Staubli VAL3: cvIn.pjx

--- cvIn.pjx ---
Parameters version=s7.6.2 stackSize=5000 millimeterUnit=true
Program file=checkTrackArea.pgx
Program file=conveyor.pgx
Program file=create.pgx
Program file=disableQueue.pgx
Program file=enableQueue.pgx
Program file=fillQueue.pgx
Program file=flushQueue.pgx
Program file=getConvFrame.pgx
Program file=getDetectDist.pgx
Program file=getDetectFrame.pgx
Program file=getDistance.pgx
Program file=getErrorMessage.pgx
Program file=getNextID.pgx
Program file=getObjectData.pgx
Program file=getObjectLatch.pgx
Program file=getObjectOffset.pgx
Program file=getObjectPos.pgx
Program file=getStatus.pgx
Program file=getTravelDist.pgx
Program file=init.pgx
Program file=kill.pgx
Program file=releaseObject.pgx
Program file=removePart.pgx
Program file=reset.pgx
Program file=setCalibrating.pgx
Program file=setConveyor.pgx
Program file=setObjectInUse.pgx
Program file=start.pgx
Program file=stop.pgx
Program file=teach.pgx
Program file=whichObjectUsed.pgx
Data file=cvIn.dtx
Library alias=cfg path=Disk://Tracking/config/config.pjx autoload=true password=
Library alias=det path=Disk://Tracking/Templates/GenericDetect/GenericDetect.pjx autoload=false password=
Library alias=enc path=Disk://Tracking/Templates/GenericEnc/GenericEnc.pjx autoload=false password=
Library alias=geometry path=Disk://Tracking/Templates/Geometry/Geometry.pjx autoload=false password=
Library alias=swap path=Disk://Tracking/Swap/Swap.pjx autoload=true password=
Library alias=ut path=Disk://Tracking/Tools/util/util.pjx autoload=true password=
Library alias=lang path=Disk://Tracking/language/english/english.pjx autoload=true password=
Library alias=out path=Disk://Tracking/io/outputs/outputs.pjx autoload=true password=

--- cvIn.dtx ---
bool bClockEnabled = true
bool bEnableQueuing = true
bool bInit = true
public bool bLOG = true
public bool bLinear = true
bool bLockQueueAcces
bool bResetConv
public bool bUseUserCenter
public bool bUseUserLimit
dio doClock = {link=BasicIO-1\%Q0}
public frame fConveyor = {x=365.904087, y=326.91934, z=-82.602337, rx=-0.010861, ry=-0.059106, rz=0.004608, fatherId=world[0]}
public frame fDetection = {x=392.598601, y=461.346273, z=-82.976862, rx=0.205045, ry=0.617271, rz=0.011036, fatherId=world[0]}
num nA1 = -1.427414
num nA2 = -1.428787
num nAddedToQueue
num nB1
num nB2 = 436.58822
num nBoundaryDwn
num nBoundaryUp
public num nBufferSize = 100
public num nCalibratedDist
num nCalibratedID = -99
public num nClockPeriod = 210
public num nConveyorSpeed = 495.277368
num nDEFAULTID = -99
num nDETECT_OVR = 11
public num nDetection2Rob = 945.961992
public num nENCRESOLUTION = 2000
public num nENCSCALEFACTOR = 0.7207
num nEncLatchedVal[100]
num nErrVal[4]
public num nFirDelay = 0.004
public num nFirOrdre = 20
num nFirTime = 0.04
num nIdxCalib
num nIdxPull
num nIdxPush
public num nLatchLockDist
num nNumbOfUser[100]
num nPUSH_NEGATIVE = 10
public num nPosMatchTol = 50
num nQueueID[100]
  [0] = -99
  [1] = -99
  [2] = -99
  [3] = -99
  [4] = -99
  [5] = -99
  [6] = -99
  [7] = -99
  [8] = -99
  [9] = -99
  [10] = -99
  [11] = -99
  [12] = -99
  [13] = -99
  [14] = -99
  [15] = -99
  [16] = -99
  [17] = -99
  [18] = -99
  [19] = -99
  [20] = -99
  [21] = -99
  [22] = -99
  [23] = -99
  [24] = -99
  [25] = -99
  [26] = -99
  [27] = -99
  [28] = -99
  [29] = -99
  [30] = -99
  [31] = -99
  [32] = -99
  [33] = -99
  [34] = -99
  [35] = -99
  [36] = -99
  [37] = -99
  [38] = -99
  [39] = -99
  [40] = -99
  [41] = -99
  [42] = -99
  [43] = -99
  [44] = -99
  [45] = -99
  [46] = -99
  [47] = -99
  [48] = -99
  [49] = -99
  [50] = -99
  [51] = -99
  [52] = -99
  [53] = -99
  [54] = -99
  [55] = -99
  [56] = -99
  [57] = -99
  [58] = -99
  [59] = -99
  [60] = -99
  [61] = -99
  [62] = -99
  [63] = -99
  [64] = -99
  [65] = -99
  [66] = -99
  [67] = -99
  [68] = -99
  [69] = -99
  [70] = -99
  [71] = -99
  [72] = -99
  [73] = -99
  [74] = -99
  [75] = -99
  [76] = -99
  [77] = -99
  [78] = -99
  [79] = -99
  [80] = -99
  [81] = -99
  [82] = -99
  [83] = -99
  [84] = -99
  [85] = -99
  [86] = -99
  [87] = -99
  [88] = -99
  [89] = -99
  [90] = -99
  [91] = -99
  [92] = -99
  [93] = -99
  [94] = -99
  [95] = -99
  [96] = -99
  [97] = -99
  [98] = -99
  [99] = -99
num nStatus
num nSysCycleTime = 0.002
num nTmpEncLatched[10]
  [0] = 4878005.31
  [1] = 4869824.31
  [2] = 4741503.57
num nTmpID[10]
  [0] = 1
  [1] = 1
  [2] = 1
public num nTrackWinHeight = 500
num nWinDownStream
num nWinUpStream
pointRs pObjectRS = {fatherId=world[0]}
pointRx pObject = {fatherId=world[0]}
public string sClockSigName = "bOut0"
string sConvNum = "CNV0"
public string sConveyorName = "cvIn"
public string sDetectionLib = "PointGrey"
public string sDwnLimSigName = "none"
public string sEncoderLib = "D_ABZ_00"
string sErrMsgList[12]
  [0] = "Success"
  [1] = "No object available (ID=*)"
  [3] = "The encoder library is not started yet."
  [4] = "The detection library is not started yet."
  [6] = "Run-time error from Conveyor library in task called *\../*. Error code is *"
  [7] = "Run-time error from Encoder library. Error code is *"
  [8] = "Run-time error from Detection library. Error code is *"
  [10] = "Warning, object with negative ID cannot be pushed into conveyor's queue"
  [11] = "Warning, detection overrun."
string sErrorMessage = "No message pending"
public string sGeometryLib = "GeometryRS"
string sMsg
string sTASK[3]
  [0] = "conveyor"
  [1] = "encoder"
  [2] = "detect"
public string sUpLimSigName = "none"
trsf trBoundaryDwn[2]
  [0] = {x=305.565702, rx=-179.989134, ry=-0.059105, rz=88.399965}
  [1] = {x=118.089887, y=267.862957, z=0.515773, rx=-179.989134, ry=-0.059105, rz=65.426002}
trsf trBoundaryUp[2]
  [0] = {rx=-179.989134, ry=-0.059105, rz=58.053225}
  [1] = {x=-187.656083, y=267.862957, rx=-179.989134, ry=-0.059105, rz=32.698528}
trsf trDEFAULT = {x=5, y=4, z=3, rx=2, ry=1}
trsf trDetectedCoord[100]
  [0] = {x=5, y=4, z=3, rx=2, ry=1}
  [1] = {x=5, y=4, z=3, rx=2, ry=1}
  [2] = {x=5, y=4, z=3, rx=2, ry=1}
  [3] = {x=5, y=4, z=3, rx=2, ry=1}
  [4] = {x=5, y=4, z=3, rx=2, ry=1}
  [5] = {x=5, y=4, z=3, rx=2, ry=1}
  [6] = {x=5, y=4, z=3, rx=2, ry=1}
  [7] = {x=5, y=4, z=3, rx=2, ry=1}
  [8] = {x=5, y=4, z=3, rx=2, ry=1}
  [9] = {x=5, y=4, z=3, rx=2, ry=1}
  [10] = {x=5, y=4, z=3, rx=2, ry=1}
  [11] = {x=5, y=4, z=3, rx=2, ry=1}
  [12] = {x=5, y=4, z=3, rx=2, ry=1}
  [13] = {x=5, y=4, z=3, rx=2, ry=1}
  [14] = {x=5, y=4, z=3, rx=2, ry=1}
  [15] = {x=5, y=4, z=3, rx=2, ry=1}
  [16] = {x=5, y=4, z=3, rx=2, ry=1}
  [17] = {x=5, y=4, z=3, rx=2, ry=1}
  [18] = {x=5, y=4, z=3, rx=2, ry=1}
  [19] = {x=5, y=4, z=3, rx=2, ry=1}
  [20] = {x=5, y=4, z=3, rx=2, ry=1}
  [21] = {x=5, y=4, z=3, rx=2, ry=1}
  [22] = {x=5, y=4, z=3, rx=2, ry=1}
  [23] = {x=5, y=4, z=3, rx=2, ry=1}
  [24] = {x=5, y=4, z=3, rx=2, ry=1}
  [25] = {x=5, y=4, z=3, rx=2, ry=1}
  [26] = {x=5, y=4, z=3, rx=2, ry=1}
  [27] = {x=5, y=4, z=3, rx=2, ry=1}
  [28] = {x=5, y=4, z=3, rx=2, ry=1}
  [29] = {x=5, y=4, z=3, rx=2, ry=1}
  [30] = {x=5, y=4, z=3, rx=2, ry=1}
  [31] = {x=5, y=4, z=3, rx=2, ry=1}
  [32] = {x=5, y=4, z=3, rx=2, ry=1}
  [33] = {x=5, y=4, z=3, rx=2, ry=1}
  [34] = {x=5, y=4, z=3, rx=2, ry=1}
  [35] = {x=5, y=4, z=3, rx=2, ry=1}
  [36] = {x=5, y=4, z=3, rx=2, ry=1}
  [37] = {x=5, y=4, z=3, rx=2, ry=1}
  [38] = {x=5, y=4, z=3, rx=2, ry=1}
  [39] = {x=5, y=4, z=3, rx=2, ry=1}
  [40] = {x=5, y=4, z=3, rx=2, ry=1}
  [41] = {x=5, y=4, z=3, rx=2, ry=1}
  [42] = {x=5, y=4, z=3, rx=2, ry=1}
  [43] = {x=5, y=4, z=3, rx=2, ry=1}
  [44] = {x=5, y=4, z=3, rx=2, ry=1}
  [45] = {x=5, y=4, z=3, rx=2, ry=1}
  [46] = {x=5, y=4, z=3, rx=2, ry=1}
  [47] = {x=5, y=4, z=3, rx=2, ry=1}
  [48] = {x=5, y=4, z=3, rx=2, ry=1}
  [49] = {x=5, y=4, z=3, rx=2, ry=1}
  [50] = {x=5, y=4, z=3, rx=2, ry=1}
  [51] = {x=5, y=4, z=3, rx=2, ry=1}
  [52] = {x=5, y=4, z=3, rx=2, ry=1}
  [53] = {x=5, y=4, z=3, rx=2, ry=1}
  [54] = {x=5, y=4, z=3, rx=2, ry=1}
  [55] = {x=5, y=4, z=3, rx=2, ry=1}
  [56] = {x=5, y=4, z=3, rx=2, ry=1}
  [57] = {x=5, y=4, z=3, rx=2, ry=1}
  [58] = {x=5, y=4, z=3, rx=2, ry=1}
  [59] = {x=5, y=4, z=3, rx=2, ry=1}
  [60] = {x=5, y=4, z=3, rx=2, ry=1}
  [61] = {x=5, y=4, z=3, rx=2, ry=1}
  [62] = {x=5, y=4, z=3, rx=2, ry=1}
  [63] = {x=5, y=4, z=3, rx=2, ry=1}
  [64] = {x=5, y=4, z=3, rx=2, ry=1}
  [65] = {x=5, y=4, z=3, rx=2, ry=1}
  [66] = {x=5, y=4, z=3, rx=2, ry=1}
  [67] = {x=5, y=4, z=3, rx=2, ry=1}
  [68] = {x=5, y=4, z=3, rx=2, ry=1}
  [69] = {x=5, y=4, z=3, rx=2, ry=1}
  [70] = {x=5, y=4, z=3, rx=2, ry=1}
  [71] = {x=5, y=4, z=3, rx=2, ry=1}
  [72] = {x=5, y=4, z=3, rx=2, ry=1}
  [73] = {x=5, y=4, z=3, rx=2, ry=1}
  [74] = {x=5, y=4, z=3, rx=2, ry=1}
  [75] = {x=5, y=4, z=3, rx=2, ry=1}
  [76] = {x=5, y=4, z=3, rx=2, ry=1}
  [77] = {x=5, y=4, z=3, rx=2, ry=1}
  [78] = {x=5, y=4, z=3, rx=2, ry=1}
  [79] = {x=5, y=4, z=3, rx=2, ry=1}
  [80] = {x=5, y=4, z=3, rx=2, ry=1}
  [81] = {x=5, y=4, z=3, rx=2, ry=1}
  [82] = {x=5, y=4, z=3, rx=2, ry=1}
  [83] = {x=5, y=4, z=3, rx=2, ry=1}
  [84] = {x=5, y=4, z=3, rx=2, ry=1}
  [85] = {x=5, y=4, z=3, rx=2, ry=1}
  [86] = {x=5, y=4, z=3, rx=2, ry=1}
  [87] = {x=5, y=4, z=3, rx=2, ry=1}
  [88] = {x=5, y=4, z=3, rx=2, ry=1}
  [89] = {x=5, y=4, z=3, rx=2, ry=1}
  [90] = {x=5, y=4, z=3, rx=2, ry=1}
  [91] = {x=5, y=4, z=3, rx=2, ry=1}
  [92] = {x=5, y=4, z=3, rx=2, ry=1}
  [93] = {x=5, y=4, z=3, rx=2, ry=1}
  [94] = {x=5, y=4, z=3, rx=2, ry=1}
  [95] = {x=5, y=4, z=3, rx=2, ry=1}
  [96] = {x=5, y=4, z=3, rx=2, ry=1}
  [97] = {x=5, y=4, z=3, rx=2, ry=1}
  [98] = {x=5, y=4, z=3, rx=2, ry=1}
  [99] = {x=5, y=4, z=3, rx=2, ry=1}
trsf trTmp[10]
  [0] = {x=-13.6, y=13.6, rz=90}
  [1] = {x=-105.5, y=-8.6, rz=91}
  [2] = {x=-185.6, y=-3.4, rz=87.4}

--- conveyor.pgx ---
program conveyor()
  local bool l_bLatched
  local bool l_bLock
  local bool l_bMemoCalib
  local num l_nDelayEnLatch
  local num l_nEncEnaLatVal
  local num l_nEncLatchVal
  local num l_nEncValue
  local num l_nLatchLocked
  local num l_nNumOfObject
  local num l_nStepFill
  local num l_nTimeLatched
  local num l_nTrigger
begin
  //
  //----------------------------------------------------------------
  l_nEncEnaLatVal=l_nEncLatchVal=l_nEncValue
  l_bMemoCalib=det:bCalibrating
  //
  //--- Enable latch feature of the encoder library
  enc:bLatchEnabled=true
  if bClockEnabled
    l_nStepFill=-1
  else
    l_nStepFill=0
  endIf
  l_nTimeLatched=clock()
  //*****
  //
  // Initializing the output to start if it's used
  if bClockEnabled
    // If position capture OUTPUT occurs on falling edge
    // CHANGE the logic of the output doClock at all lines of this program.
    // false-->true / true-->false
    doClock=false
  endIf
  // waiting the task's detection is running
  wait(det:bTaskDetOK)
  //****   MAIN LOOP
  while true
    //--- Read instantaneous encoder value
    l_nEncValue=aioGet(enc:aiEncCurrentPos)
    //
    //*****  CLOCK SECTION
    l_nLatchLocked=sel(bClockEnabled,max(2*nClockPeriod/3,nLatchLockDist),nLatchLockDist)
    // Check if feature is enabled
    if bClockEnabled
      // If trigger OFF, and If the conveyor has moved more than the trigger perriod
      if (doClock==false) and abs((l_nEncValue-l_nEncEnaLatVal)*nENCSCALEFACTOR)>nClockPeriod
        // If system ready, set trigger
        // Else, set Status in overrun
        if l_nStepFill==-1
          l_nStepFill=0
          doClock=true
          l_nTrigger=l_nTrigger+1
          logMsg("trigger num: "+toString("",l_nTrigger)+" :"+toString("0.2",clock())+" s")
          logMsg("trigger: "+toString(".2",(l_nEncValue-l_nEncEnaLatVal)*nENCSCALEFACTOR)+" mm")
          l_nEncEnaLatVal=l_nEncValue
          if bAnd(cfg:nLog,cfg:nLOGDETECT)==cfg:nLOGDETECT and bLOG
            ? sConvNum+"(conveyor)>>Set trigger. Clock :"+toString(".2",clock())
          endIf
        elseIf nStatus!=2
          // Warning, detection overrun. Object(s) wont been queued
          if bAnd(cfg:nLog,cfg:nLOGDETECT)==cfg:nLOGDETECT and bLOG
            ? sConvNum+"(conveyor)>>Detection Overrun : Cannot set trigger on time. Clock :"+toString(".2",clock())
          endIf
          nStatus=2
          sErrorMessage=sErrMsgList[nDETECT_OVR]
        endIf
      endIf
      // If trigger ON, and If the conveyor has move more than half of the trigger period
      // reset trigger
      if (doClock==true) and abs((l_nEncValue-l_nEncEnaLatVal)*nENCSCALEFACTOR)>nClockPeriod/2
        doClock=false
      endIf
    endIf
    //
    //*****  CONVEYOR SECTION
    if left(sDetectionLib,6)=="Socket" and !det:bCalibrating
      // When working with the detection library "Socket" and the conveyor
      //  isn't calibrating the distance from the sensor, the encoder
      //  latched value is given by the "Socket" and the encoder library is
      //  not used.
      l_bLatched=true
      l_nEncLatchVal=0
      if l_nStepFill==0
        l_nStepFill=1
      endIf
    else
      // Reinitialize conveyor sequence when detection library "Socket"
      //  goes into Calibration Mode.
      if left(sDetectionLib,6)=="Socket" and det:bCalibrating and !l_bMemoCalib
        l_nStepFill=0
        det:nNumOfPart=-1
      endIf
      // Use the encoder library to get the encoder latched value.
      // Check if latch occured
      call enc:isLatched(l_bLatched)
      // If part latched, get encoder latched value.
      // Else, re-enable latching at the encoder library
      if l_bLatched==true
        logMsg("getLatched: "+toString(".2",clock())+" s")
        det:nNumOfPart=-1
        delay(0)
        call enc:resetLatch()
        if bAnd(cfg:nLog,cfg:nLOGDETECT)==cfg:nLOGDETECT and bLOG
          ? sConvNum+"(conveyor)>>Object latched detected. Clock :"+toString(".2",clock())
        endIf
        //
        // Start timer for re-enabling latch feature
        l_nDelayEnLatch=clock()
        //
        // If system ready, get encoder latched value.
        // Else, overrun for external latch
        if l_nStepFill==0
          l_nStepFill=1
          l_bLock=false
          // Get encoder latched value
          call enc:getValue(true,l_nEncLatchVal)
          // Disable latch feature of the encoder library until conveyor has moved
          // the distance defined by the user (variable nLatchLockDist)
          enc:bLatchEnabled=false
          // Record clock of Latch
          l_nTimeLatched=clock()
          //
          //Overrun for external latch
        elseIf !bClockEnabled and nStatus!=2
          // Warning, detection overrun. Object(s) wont been queued
          if bAnd(cfg:nLog,cfg:nLOGDETECT)==cfg:nLOGDETECT and bLOG
            ? sConvNum+"(conveyor)>>Detection Overrun : System not ready to latch again."
          endIf
          nStatus=2
          sErrorMessage=sErrMsgList[nDETECT_OVR]
        endIf
      else
        // wait a while before re-enabling the latch feature
        if clock()-l_nDelayEnLatch>0.02
          // Latch feature not enabled
          if (enc:bLatchEnabled==false)
            // Check conveyor's advance
            if abs((l_nEncValue-l_nEncLatchVal)*nENCSCALEFACTOR)>=l_nLatchLocked
              enc:bLatchEnabled=true
            endIf
          endIf
        endIf
      endIf
    endIf
    l_bMemoCalib=det:bCalibrating
    //
    //--- Poll detection library
    if bEnableQueuing==true
      switch l_nStepFill
        // Poll detection lib for number of detected objects
        case 1
          if l_bLock==false
            if bAnd(cfg:nLog,cfg:nLOGDETECT)==cfg:nLOGDETECT and bLOG
              ? sConvNum+"(conveyor)>>Reading number of detected objects"
            endIf
            l_bLock=true
          endIf
          //
          if l_bLock==true
            call det:isDetected(l_nNumOfObject)
            if (l_nNumOfObject>=0)
              l_nStepFill=sel(l_nNumOfObject>0,10,20)
              l_bLock=false
            endIf
          endIf
        break
        // Queue detected objects
        case 10
          if l_bLock==false
            if bAnd(cfg:nLog,cfg:nLOGDETECT)==cfg:nLOGDETECT and bLOG
              ? sConvNum+"(conveyor)>>Response time of the detection lib: "+toString(".2",clock()-l_nTimeLatched)+" sec."
            endIf
            call fillQueue(l_nNumOfObject,l_nEncLatchVal)
            l_bLock=true
          endIf
          if l_bLock==true
            l_nStepFill=20
            l_bLock=false
          endIf
        break
        // Acknowledge detection library
        case 20
          if l_bLock==false
            if bAnd(cfg:nLog,cfg:nLOGDETECT)==cfg:nLOGDETECT and bLOG
              ? sConvNum+"(conveyor)>>Reset nNumOfPart variable of detection lib"
            endIf
            //det:nNumOfPart=-1
            if nStatus==2
              if bAnd(cfg:nLog,cfg:nLOGDETECT)==cfg:nLOGDETECT and bLOG
                ? sConvNum+"(conveyor)>>Detection Overrun : Time to recover data after latch :"+toString(".2",clock()-l_nTimeLatched)+" sec."
              endIf
              nStatus=0
            endIf
            if bClockEnabled
              l_nStepFill=-1
            else
              l_nStepFill=0
            endIf
          endIf
        break
      endSwitch
    endIf
    //
    // //*****  RESET SECTION
    if bResetConv==true
      call flushQueue()
      bResetConv=false
    endIf
    //
    delay(0)
  endWhile
end

--- getDetectFrame.pgx ---
public program getDetectFrame(frame& x_fDetection (dimensions=1), frame x_fRefFrame (dimensions=1), num& x_nError (dimensions=1))
  local string l_sCustomTxt[2]
begin
  // This program returns the position of the conveyor frame
  // in the réference frame passed as parameter
  //
  // Input param
  //  x_fRefFrame   : Reference frame in which the position of the conveyor
  //                frame must be returned
  //
  // Output param
  //  x_fConveyor   : Conveyor frame
  //  x_nError      : Error code
  //    0    --> No error
  //    14   --> Conveyor library not started, the frame cannot be computed.
  //
  // Created 7-03-08                                   C.CURRIVAND
  //----------------------------------------------------------------
  x_nError=0
  if bInit
    x_fDetection.trsf=position(fDetection,x_fRefFrame)
  else
    x_nError=14
    // Prepare clear text error message
    l_sCustomTxt[0]=sConveyorName
    l_sCustomTxt[1]="detection"
    call ut:addStrToString(lang:sListOfMessage[x_nError],sErrorMessage,"",l_sCustomTxt)
  endIf
end

--- getStatus.pgx ---
public program getStatus(num x_nConvNum (dimensions=1), num& x_nStatus[] (dimensions=1))
  local bool l_bLock
  local bool l_bQuit
  local num l_i
  local num l_nStatus
  local num l_nStep
  local string l_sSubString
begin
  // This program returns the status of the conveyor library
  //
  // Input Param
  // x_nConvNum    : Conveyor Number
  //
  // Output Param
  //  x_nStatus    : Status of the conveyor library
  //
  //Created 04-06-07                              C.CURRIVAND
  //--------------------------------------------------------------
  //
  l_bQuit=false
  do
    switch l_nStep
      // Check status of the encoder library
      case 0
        call enc:getStatus(l_nStatus)
        if (l_nStatus!=0)
          // Prepare clear text error message
          call ut:addNumToString(sErrMsgList[7],sErrorMessage,"",l_nStatus)
          l_bQuit=true
        else
          l_nStep=20
        endIf
      break
      // Check status of the detection library.
      case 10
        //call det:getStatus(l_nStatus)
        if (l_nStatus!=0)
          // Prepare clear text error message
          call ut:addNumToString(sErrMsgList[8],sErrorMessage,"",l_nStatus)
          l_bQuit=true
        else
          l_nStep=20
        endIf
      break
      // check status of the conveyor task
      // sTASK[0]=conveyor
      case 20
        l_nStatus=taskStatus(sTASK[0]+toString("",x_nConvNum))
        if (l_nStatus!=0) and (l_nStatus!=1)
          // Prepare clear text error message
          if l_nStatus==-1
            // Task not created (yet !)
            l_nStatus=2999
          else
            // Run-time error
            l_nStatus=2000+l_nStatus
          endIf
          l_sSubString=sTASK[0]+toString("",x_nConvNum)
          call ut:addStrToString(sErrMsgList[6],sErrorMessage,"",l_sSubString)
          call ut:addNumToString(sErrorMessage,sErrorMessage,"*",l_nStatus)
          l_bQuit=true
        endIf
        if (l_nStatus==0) or (l_nStatus==1)
          l_nStatus=nStatus
          nStatus=0
        endIf
        l_bQuit=true
      break
    endSwitch
    delay(0)
  until l_bQuit==true
  x_nStatus=l_nStatus
end

--- getTravelDist.pgx ---
program getTravelDist(num x_nIdx (dimensions=1), num& x_nTravelDist[] (dimensions=1), num& x_nError[] (dimensions=1))
  local num l_nEncValue
begin
  // This program returns the distance between the instantaneous
  // conveyor's position and the one when it was last latched.
  //
  // Input param
  //  x_nIdx    : Index of the object in the queue
  //
  // Output param
  //  x_nTravelDist : Distance
  //  x_nError      : Error code
  //    0 : No error
  //    1 : No object available
  //
  //----------------------------------------------------------------
  //
  x_nError=0
  if nNumbOfUser[x_nIdx]!=0
    l_nEncValue=aioGet(enc:aiEncCurrentPos)
    // Test for encoder roll over
    if l_nEncValue<nEncLatchedVal[x_nIdx]
      // roll over
      x_nTravelDist=nENCSCALEFACTOR*(enc:nMAXCOUNT-nEncLatchedVal[x_nIdx]+l_nEncValue-enc:nMINCOUNT)
    else
      // No roll over
      x_nTravelDist=nENCSCALEFACTOR*(l_nEncValue-nEncLatchedVal[x_nIdx])
    endIf
  else
    //* No Object requested
    x_nError=1
    if cfg:bLog==true
      nErrVal[0]=x_nIdx
      call ut:addNumToString(sConvNum+"(getTravelDist)>>:"+sErrMsgList[x_nError],sMsg,"*",nErrVal)
      logMsg(sMsg)
    endIf
  endIf
end

--- teach.pgx ---
public program teach(tool x_tTool (dimensions=1), frame x_fFrame (dimensions=1), point& x_pLoc[] (dimensions=1), num& x_nError[] (dimensions=1))
  local bool l_bExit
  local bool l_bFound
  local num l_i
  local num l_nError
  local num l_nObjectOffset
  local string l_str
begin
  // This program records the encoder offset associated with the
  // object, which ID is given by the detection Library. This encoder offset
  // is used as reference to evaluate the shifting of the object laying
  // on the conveyor.The program memorizes which object ID have been already
  // calibrated
  //
  // Input Param
  //  x_tTool   : Tool for motion
  //  x_fFrame  : Reference frame in which the location must be taught
  //
  // Output Param
  // x_pLoc   : Taught location
  // x_nError : Error code
  //    =0    : No error
  //    =-1   : No object detected, not possible to teach anything
  //
  // Created 11-01-06                                   C.CURRIVAND
  //----------------------------------------------------------------
  //
  // Initialisations
  x_nError=0
  l_bExit=false
  l_bFound=false
  // Check if an object has been detected
  if nNumbOfUser[nIdxPull]!=0
    nIdxCalib=0
    if bAnd(cfg:nLog,cfg:nLOGMISC)==cfg:nLOGMISC
      ? sConvNum+"(teach)>>CALIBRATING ID "+toString("",nQueueID[nIdxPull])
    endIf
    do
      if bAnd(cfg:nLog,cfg:nLOGMISC)==cfg:nLOGMISC
        l_str=sConvNum+"(teach)>>CalibratedID["+toString("",nIdxCalib)+"]: "+toString("",nCalibratedID[nIdxCalib])
        l_str=l_str+"  DetectedID: "+toString("",nQueueID[nIdxPull])
        l_str=l_str+"  CalibratedDist["+toString("",nIdxCalib)+"]: "+toString("",nCalibratedDist[nIdxPull])
        ? l_str
      endIf
      // Check if ID has already been calibrated
      l_bFound=(nCalibratedID[nIdxCalib]==nDEFAULTID) or (nQueueID[nIdxPull]==nCalibratedID[nIdxCalib])
      if !l_bFound
        nIdxCalib=nIdxCalib+1
        l_bExit=(nIdxCalib>=size(nCalibratedID))
      endIf
    until l_bExit or l_bFound
    //
    // The object has not been calibrated (yet!)
    if !l_bFound
      if bAnd(cfg:nLog,cfg:nLOGMISC)==cfg:nLOGMISC
        logMsg(sConvNum+"(teach)>>Object with ID "+toString("",nQueueID[nIdxPull])+" has never been calibrated,add to list")
      endIf
      resize(nCalibratedID,1,size(nCalibratedID)+1)
      resize(nCalibratedDist,1,size(nCalibratedDist)+1)
      // update data
      nCalibratedID[nIdxCalib]=nQueueID[nIdxPull]
      nCalibratedDist[nIdxCalib]=nENCSCALEFACTOR*(aioGet(enc:aiEncCurrentPos)-nEncLatchedVal[nIdxPull])-nDetection2Rob
      l_nObjectOffset=0
    else
      // this object has aready been calibrated, compute offset between current position
      // and position when it has been calibrated
      if bAnd(cfg:nLog,cfg:nLOGMISC)==cfg:nLOGMISC
        ? sConvNum+"(teach)>>Object with ID "+toString("",nQueueID[nIdxPull])+" is calibrated"
      endIf
      call getObjectOffset(nIdxPull,l_nObjectOffset,l_nError)
    endIf
    // returns robot position
    x_pLoc.trsf=position(compose(here(x_tTool,world),fConveyor,{-l_nObjectOffset,0,0,0,0,0}),x_fFrame)
    //
    // saving data
    x_nError=libSave()
    if bAnd(cfg:nLog,cfg:nLOGMISC)==cfg:nLOGMISC
      if x_nError==0
        ? sConvNum+"(teach)>>Calibration data for ID "+toString("",nQueueID[nIdxPull])+" saved successfully"
      else
        ? sConvNum+"(teach)>>ERROR "+toString("",x_nError)+" while saving data for ID "+toString("",x_nError)
      endIf
    endIf
  else
    x_nError=-1
    if bAnd(cfg:nLog,cfg:nLOGMISC)==cfg:nLOGMISC
      ? sConvNum+"(teach)>>No object detected for teaching"
    endIf
  endIf
end
